PROGRAM MAIN
VAR
END_VAR

END_PROGRAM

(* stored: Version 1.1.0.1
   POU MAIN: Id {c596badd-3279-4066-b122-ed8d929cff95} *)
